{attribute 'qualified_only'}
TYPE E_AutoOffOn :
(
	_invalid := 0,
	
	Auto := 1,
	Off := 2,
	On := 3
) UDINT;
END_TYPE

(* stored: Version 1.1.0.1
   DUT E_AutoOffOn: Id {e9208f05-3f69-4706-9f16-6b581ca68387} *)
